// TIA Portal V19 export
DATA_BLOCK "EnS_Org_CycInt500ms"   // DB3
TITLE = Instance DB of organizational data in cyclic interrupt OB
// Instance DB of organizational data in cyclic interrupt OB
// stored: InstanceOfName EnS_Organization, InstanceOfType FB
"EnS_Organization"
   // VAR_INPUT
   //    runUpCyc { ExternalAccessible := 'False'; ExternalVisible := 'False'; ExternalWritable := 'False'} : UInt := 20;
   //    messageSuppress { ExternalAccessible := 'False'; ExternalVisible := 'False'; ExternalWritable := 'False'} : Bool;
   // END_VAR
   // VAR_OUTPUT
   //    orgData { ExternalAccessible := 'False'; ExternalVisible := 'False'; ExternalWritable := 'False'} : "EnS_typeOrgData";
   // END_VAR
   // VAR
   //    su16_RunUpCyc { ExternalAccessible := 'False'; ExternalVisible := 'False'; ExternalWritable := 'False'} : UInt;
   // END_VAR
BEGIN
END_DATA_BLOCK
